# EPICS autosave request: FOFBApp/Db/FOFBInfo_settings.req
$(P)$(R)INFOTBTRate-SP
$(P)$(R)INFOFOFBRate-SP
$(P)$(R)INFOMONITRate-SP
$(P)$(R)INFOMONIT1Rate-SP
